PROGRAM MAIN
VAR
	En:BOOL;
	Shot:BOOL;
	Result:ARRAY [0..7] OF REAL;
END_VAR

Motion.InitMotion();
GVL.Vision();

MedidaTemp();

OperatingModes();

IF GVL.Mode = Modes.AUTO THEN
	Basic();
END_IF

Manual();
VisuLogic();
Motion();

END_PROGRAM

(* stored: Version 1.1.0.1, ProductVersion 3.1.4024.9
   POU MAIN: Id {d8de5791-f153-470a-bfaa-453c619a7f06}, SpecialFunc None *)
